# EPICS substitutions: db/ecmcEL5101.substitutions
# All fields related to postion scaling and alarms
file ecmcEcSlave.template
{
  pattern {}
          {}
}

file ecmcEL5101.template
{
    pattern {LINR,    ESLO,   EOFF,   EGU,        PREC, LOW, LOLO, HIGH, HIHI, HYST, LLSV,       LSV,        HSV,        HHSV      }
            {"SLOPE", 1,      0,      "Steps",    0,    0,   0,    0,    0,    0,    "NO_ALARM", "NO_ALARM", "NO_ALARM", "NO_ALARM"}
}
